Staubli VAL3: IOModule.pjx

Parameters version=s7.7.2 stackSize=5000 millimeterUnit=true
Program file=init.pgx
Program file=start.pgx
Program file=stop.pgx
Data file=IOModule.dtx
